{attribute 'qualified_only'}
VAR_GLOBAL

END_VAR

(* stored: Version 1.1.0.1, ProductVersion 3.1.4022.18
   GVL TransportSystemIO: Id {36f583f3-394d-4f30-a02f-925b3f63423e} *)
